PROGRAM Init
VAR
END_VAR

// Write your init sequence here

END_PROGRAM

(* stored: Version 1.1.0.1, ProductVersion 3.1.4022.18
   POU Init: Id {9544ebca-da74-4df8-a5ce-83c5c3b96401}, SpecialFunc None *)
